// TIA Portal V17 export
// export: Created 2025-05-22T06:01:50.2923024Z, ExportSetting WithDefaults, DisplayName Totally Integrated Automation Portal, DisplayVersion V17 Update 8, DisplayName TIA Portal Openness, DisplayVersion V17 Update 8, DisplayName TIA Portal Version Control Interface, DisplayVersion V17, DisplayName SINAMICS Startdrive Advanced, DisplayVersion V17 SP2, DisplayName SINAMICS Startdrive G110M, G120, G120C, G120D, G120P, G115D, DisplayVersion V17 SP2, DisplayName SINAMICS Startdrive G130, G150, S120, S150, SINAMICS MV, S210, DisplayVersion V17 SP2, DisplayName STEP 7 Professional, DisplayVersion V17 Update 8, DisplayName SINUMERIK ONE STEP 7 Toolbox, DisplayVersion V17 Update 12, DisplayName SINUMERIK ONE PLC Basic Program Plus, DisplayVersion V17 Update 12, DisplayName SINUMERIK 840D sl STEP 7 Toolbox, DisplayVersion V17 Update 12, DisplayName STEP 7 Safety, DisplayVersion V17 Update 6, DisplayName WinCC Advanced, DisplayVersion V17 Update 8
FUNCTION_BLOCK "FB2006_REFERENCE_MODE"   // FB2006, LAD
{ S7_Optimized_Access := 'FALSE' }
VERSION : 0.1
// stored: AutoNumber false, IsIECCheckEnabled false, SetENOAutomatically false, UDAEnableTagReadback false
   VAR_INPUT
      ENABLE_REQ { ExternalAccessible := 'False'; ExternalVisible := 'False'; ExternalWritable := 'False'} : Bool;   // ENABLE_REQUEST
      DISABLE_REQ { ExternalAccessible := 'False'; ExternalVisible := 'False'; ExternalWritable := 'False'} : Bool;   // DISABLE_REQUEST
   END_VAR
   VAR_OUTPUT
      REF_MODE_SLCTD_WRN { ExternalAccessible := 'False'; ExternalVisible := 'False'; ExternalWritable := 'False'} : Bool;   // REFERENCE MODE SELECTED WARNING
   END_VAR
   VAR_IN_OUT
      MODE_GROUP_DB : Struct   // MODE GROUP DB
         GENERAL : "AUTO_SINGLE_SEMI_MANUAL";
         STEP_BY_STEP : "MODES";
         MDA : "MODES";
         REFERENCE : "MODES";
         INCREMENTAL : "INCREMENTAL";
         BA : "BA_MODE";
      END_STRUCT;
   END_VAR
   VAR_TEMP
      DB_NUMBER : DInt;   // DB NUMBER FOR ALARM DECODING
   END_VAR
   // // MODE_GROUP_DB.STEP_BY_STEP.MODE_SELECTED : STEP BY STEP MODE SELECTED
   // // MODE_GROUP_DB.MDA.MODE_SELECTED : MDA MODE SELECTED
   // // MODE_GROUP_DB.REFERENCE.MODE_SELECTED : REFERENCE MODE SELECTED
   VAR_TEMP   // added for the SCL form of the ladder/FBD networks
      _w1 : Bool;
      _w2 : Bool;
   END_VAR
BEGIN

NETWORK
TITLE = READ INSTANCE DB
      L     DINO;
      +     10#800000;
      T     #DB_NUMBER;


REGION Network 2: GENERAL CONDITIONS
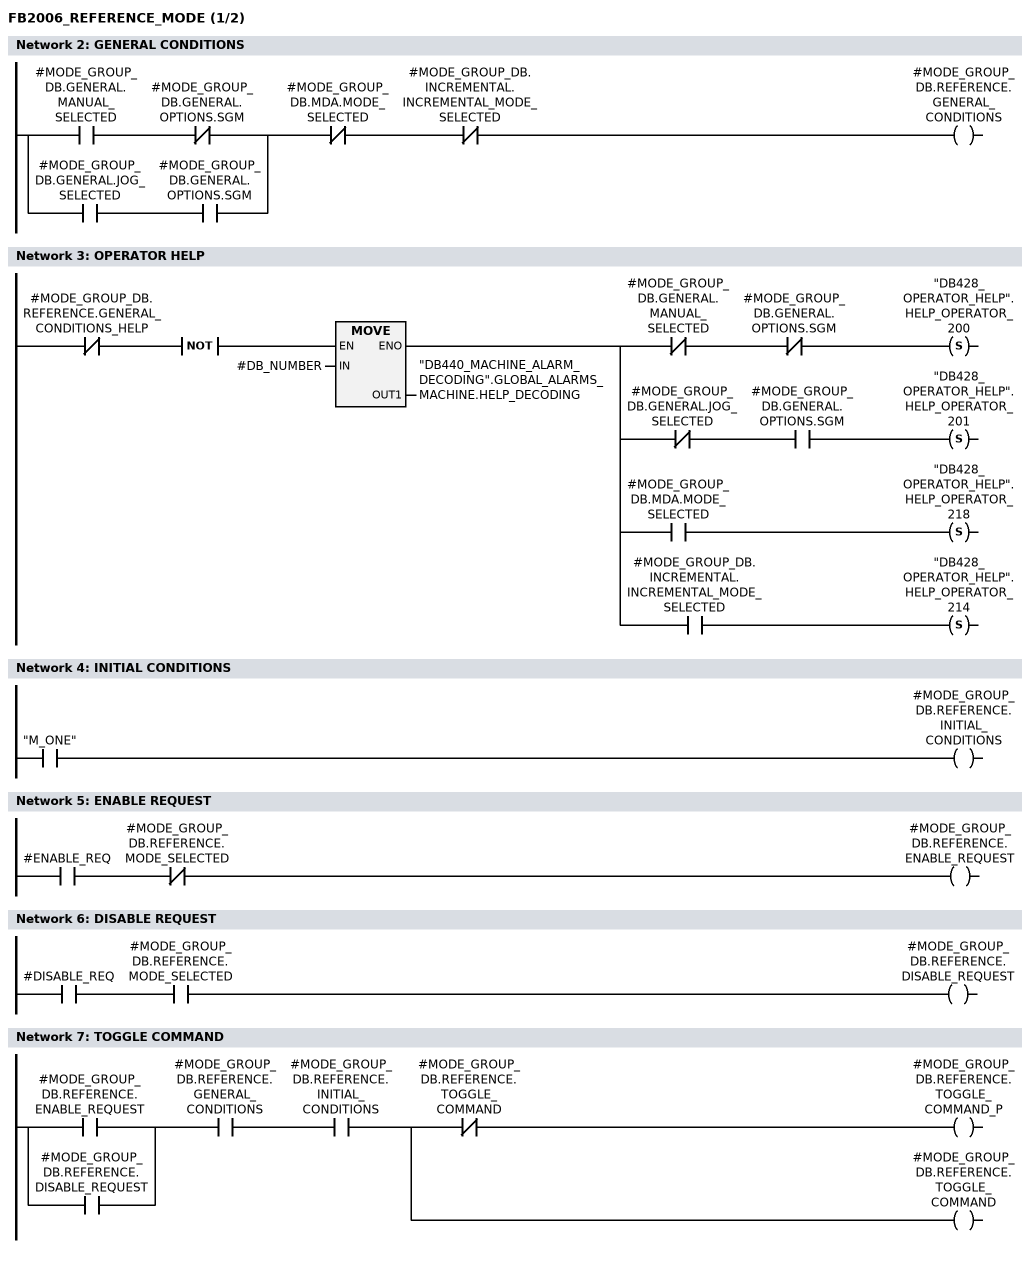
   RUNG wire#powerrail
      Contact( #MODE_GROUP_DB.GENERAL.MANUAL_SELECTED )
      I_Contact( #MODE_GROUP_DB.GENERAL.OPTIONS.SGM )
      wire#w1
      I_Contact( #MODE_GROUP_DB.MDA.MODE_SELECTED )
      I_Contact( #MODE_GROUP_DB.INCREMENTAL.INCREMENTAL_MODE_SELECTED )
      Coil( #MODE_GROUP_DB.REFERENCE.GENERAL_CONDITIONS )
   END_RUNG
   RUNG wire#powerrail
      Contact( #MODE_GROUP_DB.GENERAL.JOG_SELECTED )
      Contact( #MODE_GROUP_DB.GENERAL.OPTIONS.SGM )
   END_RUNG wire#w1
   // the same network as SCL:
   #MODE_GROUP_DB.REFERENCE.GENERAL_CONDITIONS := ((#MODE_GROUP_DB.GENERAL.MANUAL_SELECTED AND NOT #MODE_GROUP_DB.GENERAL.OPTIONS.SGM) OR (#MODE_GROUP_DB.GENERAL.JOG_SELECTED AND #MODE_GROUP_DB.GENERAL.OPTIONS.SGM)) AND NOT #MODE_GROUP_DB.MDA.MODE_SELECTED AND NOT #MODE_GROUP_DB.INCREMENTAL.INCREMENTAL_MODE_SELECTED;
END_REGION

REGION Network 3: OPERATOR HELP
   RUNG wire#powerrail
      I_Contact( #MODE_GROUP_DB.REFERENCE.GENERAL_CONDITIONS_HELP )
      Not()
      { S7_GenerateENO := "TRUE" } Move(in := #DB_NUMBER, out1 => "DB440_MACHINE_ALARM_DECODING".GLOBAL_ALARMS_MACHINE.HELP_DECODING)
      wire#w1
      I_Contact( #MODE_GROUP_DB.GENERAL.MANUAL_SELECTED )
      I_Contact( #MODE_GROUP_DB.GENERAL.OPTIONS.SGM )
      S_Coil( "DB428_OPERATOR_HELP".HELP_OPERATOR_200 )
   END_RUNG
   RUNG wire#w1
      I_Contact( #MODE_GROUP_DB.GENERAL.JOG_SELECTED )
      Contact( #MODE_GROUP_DB.GENERAL.OPTIONS.SGM )
      S_Coil( "DB428_OPERATOR_HELP".HELP_OPERATOR_201 )
   END_RUNG
   RUNG wire#w1
      Contact( #MODE_GROUP_DB.MDA.MODE_SELECTED )
      S_Coil( "DB428_OPERATOR_HELP".HELP_OPERATOR_218 )
   END_RUNG
   RUNG wire#w1
      Contact( #MODE_GROUP_DB.INCREMENTAL.INCREMENTAL_MODE_SELECTED )
      S_Coil( "DB428_OPERATOR_HELP".HELP_OPERATOR_214 )
   END_RUNG
   // the same network as SCL:
   // ENO of a box is taken as its EN; it also drops when the box reports an error
   #_w1 := NOT (NOT #MODE_GROUP_DB.REFERENCE.GENERAL_CONDITIONS_HELP);
   IF #_w1 THEN "DB440_MACHINE_ALARM_DECODING".GLOBAL_ALARMS_MACHINE.HELP_DECODING := #DB_NUMBER; END_IF;
   IF #_w1 AND NOT #MODE_GROUP_DB.GENERAL.MANUAL_SELECTED AND NOT #MODE_GROUP_DB.GENERAL.OPTIONS.SGM THEN
       "DB428_OPERATOR_HELP".HELP_OPERATOR_200 := TRUE;
   END_IF;
   IF #_w1 AND NOT #MODE_GROUP_DB.GENERAL.JOG_SELECTED AND #MODE_GROUP_DB.GENERAL.OPTIONS.SGM THEN
       "DB428_OPERATOR_HELP".HELP_OPERATOR_201 := TRUE;
   END_IF;
   IF #_w1 AND #MODE_GROUP_DB.MDA.MODE_SELECTED THEN "DB428_OPERATOR_HELP".HELP_OPERATOR_218 := TRUE; END_IF;
   IF #_w1 AND #MODE_GROUP_DB.INCREMENTAL.INCREMENTAL_MODE_SELECTED THEN
       "DB428_OPERATOR_HELP".HELP_OPERATOR_214 := TRUE;
   END_IF;
END_REGION

REGION Network 4: INITIAL CONDITIONS
   RUNG wire#powerrail
      Contact( "M_ONE" )
      Coil( #MODE_GROUP_DB.REFERENCE.INITIAL_CONDITIONS )
   END_RUNG
   // the same network as SCL:
   #MODE_GROUP_DB.REFERENCE.INITIAL_CONDITIONS := "M_ONE";
END_REGION

REGION Network 5: ENABLE REQUEST
   RUNG wire#powerrail
      Contact( #ENABLE_REQ )
      I_Contact( #MODE_GROUP_DB.REFERENCE.MODE_SELECTED )
      Coil( #MODE_GROUP_DB.REFERENCE.ENABLE_REQUEST )
   END_RUNG
   // the same network as SCL:
   #MODE_GROUP_DB.REFERENCE.ENABLE_REQUEST := #ENABLE_REQ AND NOT #MODE_GROUP_DB.REFERENCE.MODE_SELECTED;
END_REGION

REGION Network 6: DISABLE REQUEST
   RUNG wire#powerrail
      Contact( #DISABLE_REQ )
      Contact( #MODE_GROUP_DB.REFERENCE.MODE_SELECTED )
      Coil( #MODE_GROUP_DB.REFERENCE.DISABLE_REQUEST )
   END_RUNG
   // the same network as SCL:
   #MODE_GROUP_DB.REFERENCE.DISABLE_REQUEST := #DISABLE_REQ AND #MODE_GROUP_DB.REFERENCE.MODE_SELECTED;
END_REGION

REGION Network 7: TOGGLE COMMAND
   RUNG wire#powerrail
      Contact( #MODE_GROUP_DB.REFERENCE.ENABLE_REQUEST )
      wire#w1
      Contact( #MODE_GROUP_DB.REFERENCE.GENERAL_CONDITIONS )
      Contact( #MODE_GROUP_DB.REFERENCE.INITIAL_CONDITIONS )
      wire#w2
      I_Contact( #MODE_GROUP_DB.REFERENCE.TOGGLE_COMMAND )
      Coil( #MODE_GROUP_DB.REFERENCE.TOGGLE_COMMAND_P )
   END_RUNG
   RUNG wire#powerrail
      Contact( #MODE_GROUP_DB.REFERENCE.DISABLE_REQUEST )
   END_RUNG wire#w1
   RUNG wire#w2
      Coil( #MODE_GROUP_DB.REFERENCE.TOGGLE_COMMAND )
   END_RUNG
   // the same network as SCL:
   #_w1 := (#MODE_GROUP_DB.REFERENCE.ENABLE_REQUEST OR #MODE_GROUP_DB.REFERENCE.DISABLE_REQUEST) AND #MODE_GROUP_DB.REFERENCE.GENERAL_CONDITIONS AND #MODE_GROUP_DB.REFERENCE.INITIAL_CONDITIONS;
   #MODE_GROUP_DB.REFERENCE.TOGGLE_COMMAND_P := #_w1 AND NOT #MODE_GROUP_DB.REFERENCE.TOGGLE_COMMAND;
   #MODE_GROUP_DB.REFERENCE.TOGGLE_COMMAND := #_w1;
END_REGION

REGION Network 8: REFERENCE MODE SELECTED
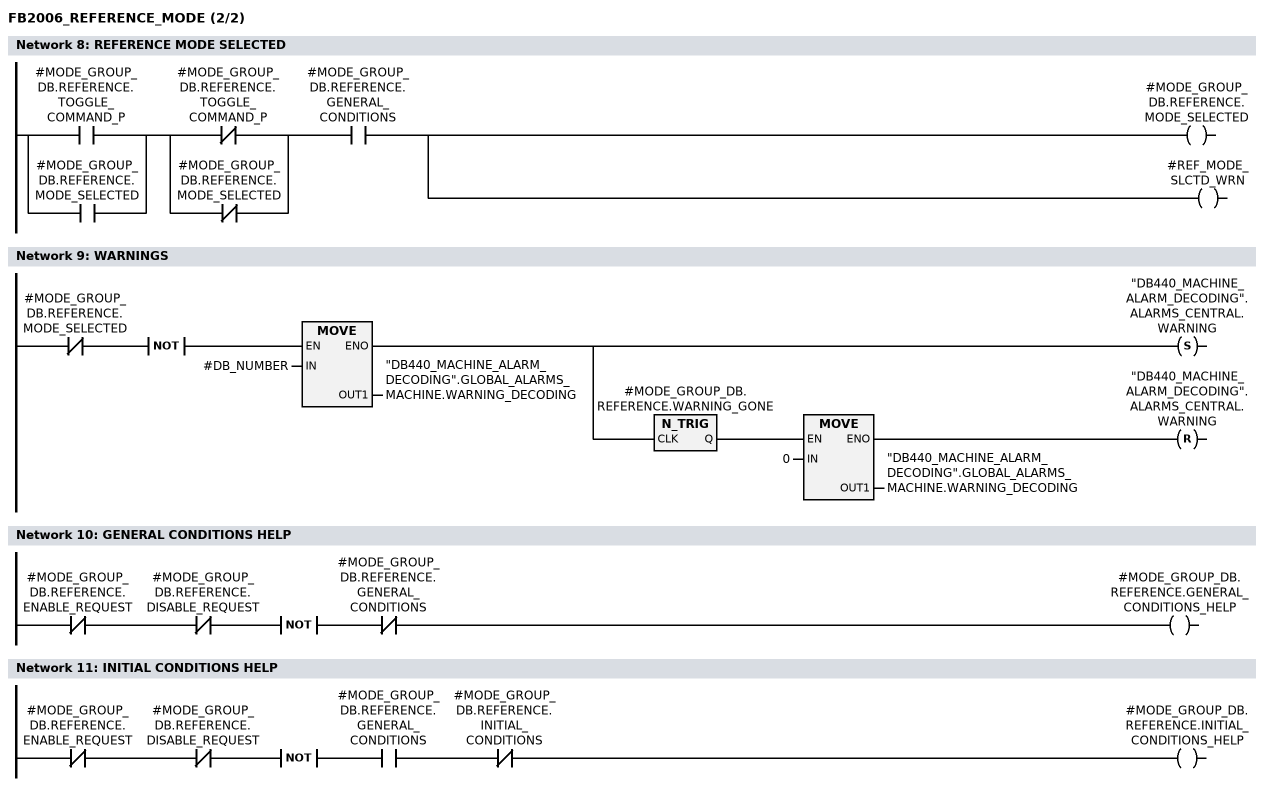
   RUNG wire#powerrail
      Contact( #MODE_GROUP_DB.REFERENCE.TOGGLE_COMMAND_P )
      wire#w1
      I_Contact( #MODE_GROUP_DB.REFERENCE.TOGGLE_COMMAND_P )
      wire#w2
      Contact( #MODE_GROUP_DB.REFERENCE.GENERAL_CONDITIONS )
      wire#w3
      Coil( #MODE_GROUP_DB.REFERENCE.MODE_SELECTED )
   END_RUNG
   RUNG wire#powerrail
      Contact( #MODE_GROUP_DB.REFERENCE.MODE_SELECTED )
   END_RUNG wire#w1
   RUNG wire#w1
      I_Contact( #MODE_GROUP_DB.REFERENCE.MODE_SELECTED )
   END_RUNG wire#w2
   RUNG wire#w3
      Coil( #REF_MODE_SLCTD_WRN )
   END_RUNG
   // the same network as SCL:
   #MODE_GROUP_DB.REFERENCE.MODE_SELECTED := (#MODE_GROUP_DB.REFERENCE.TOGGLE_COMMAND_P OR #MODE_GROUP_DB.REFERENCE.MODE_SELECTED) AND (NOT #MODE_GROUP_DB.REFERENCE.TOGGLE_COMMAND_P OR NOT #MODE_GROUP_DB.REFERENCE.MODE_SELECTED) AND #MODE_GROUP_DB.REFERENCE.GENERAL_CONDITIONS;
   #REF_MODE_SLCTD_WRN := #MODE_GROUP_DB.REFERENCE.MODE_SELECTED;
END_REGION

REGION Network 9: WARNINGS
   RUNG wire#powerrail
      I_Contact( #MODE_GROUP_DB.REFERENCE.MODE_SELECTED )
      Not()
      Move(in := #DB_NUMBER, out1 => "DB440_MACHINE_ALARM_DECODING".GLOBAL_ALARMS_MACHINE.WARNING_DECODING)
      wire#w1
      S_Coil( "DB440_MACHINE_ALARM_DECODING".ALARMS_CENTRAL.WARNING )
   END_RUNG
   RUNG wire#w1
      N_Trig( #MODE_GROUP_DB.REFERENCE.WARNING_GONE )
      Move(in := 0, out1 => "DB440_MACHINE_ALARM_DECODING".GLOBAL_ALARMS_MACHINE.WARNING_DECODING)
      R_Coil( "DB440_MACHINE_ALARM_DECODING".ALARMS_CENTRAL.WARNING )
   END_RUNG
   // the same network as SCL:
   #_w1 := NOT (NOT #MODE_GROUP_DB.REFERENCE.MODE_SELECTED);
   IF #_w1 THEN
       "DB440_MACHINE_ALARM_DECODING".GLOBAL_ALARMS_MACHINE.WARNING_DECODING := #DB_NUMBER;
       "DB440_MACHINE_ALARM_DECODING".ALARMS_CENTRAL.WARNING := TRUE;
   END_IF;
   #_w2 := NOT #_w1 AND #MODE_GROUP_DB.REFERENCE.WARNING_GONE;   // falling edge
   #MODE_GROUP_DB.REFERENCE.WARNING_GONE := #_w1;
   IF #_w2 THEN
       "DB440_MACHINE_ALARM_DECODING".GLOBAL_ALARMS_MACHINE.WARNING_DECODING := 0;
       "DB440_MACHINE_ALARM_DECODING".ALARMS_CENTRAL.WARNING := FALSE;
   END_IF;
END_REGION

REGION Network 10: GENERAL CONDITIONS HELP
   RUNG wire#powerrail
      I_Contact( #MODE_GROUP_DB.REFERENCE.ENABLE_REQUEST )
      I_Contact( #MODE_GROUP_DB.REFERENCE.DISABLE_REQUEST )
      Not()
      I_Contact( #MODE_GROUP_DB.REFERENCE.GENERAL_CONDITIONS )
      Coil( #MODE_GROUP_DB.REFERENCE.GENERAL_CONDITIONS_HELP )
   END_RUNG
   // the same network as SCL:
   #MODE_GROUP_DB.REFERENCE.GENERAL_CONDITIONS_HELP := NOT (NOT #MODE_GROUP_DB.REFERENCE.ENABLE_REQUEST AND NOT #MODE_GROUP_DB.REFERENCE.DISABLE_REQUEST) AND NOT #MODE_GROUP_DB.REFERENCE.GENERAL_CONDITIONS;
END_REGION

REGION Network 11: INITIAL CONDITIONS HELP
   RUNG wire#powerrail
      I_Contact( #MODE_GROUP_DB.REFERENCE.ENABLE_REQUEST )
      I_Contact( #MODE_GROUP_DB.REFERENCE.DISABLE_REQUEST )
      Not()
      Contact( #MODE_GROUP_DB.REFERENCE.GENERAL_CONDITIONS )
      I_Contact( #MODE_GROUP_DB.REFERENCE.INITIAL_CONDITIONS )
      Coil( #MODE_GROUP_DB.REFERENCE.INITIAL_CONDITIONS_HELP )
   END_RUNG
   // the same network as SCL:
   #MODE_GROUP_DB.REFERENCE.INITIAL_CONDITIONS_HELP := NOT (NOT #MODE_GROUP_DB.REFERENCE.ENABLE_REQUEST AND NOT #MODE_GROUP_DB.REFERENCE.DISABLE_REQUEST) AND #MODE_GROUP_DB.REFERENCE.GENERAL_CONDITIONS AND NOT #MODE_GROUP_DB.REFERENCE.INITIAL_CONDITIONS;
END_REGION
END_FUNCTION_BLOCK
